FUNCTION_BLOCK FB_ReversingSequence EXTENDS FB_CyclicFB IMPLEMENTS I_MotionSequence
VAR
	_Axis		 : I_BasicAxis;
	_Position1	 : LREAL;
	_Position2	 : LREAL;
	_Velocity	 : LREAL;
	_IdleTime	 : INT;
	fbMove		 : MC_MoveAbsolute;
	fbIdle		 : TON;
	SequenceStep : E_RevSeq;
END_VAR

{warning 'add property implementation'}
PROPERTY Axis : SPT_Motion_Control.I_BasicAxis
GET
Axis := _Axis;
END_GET
SET
_Axis := Axis;
END_SET
END_PROPERTY

{warning 'add method implementation '}
METHOD CyclicLogic
CASE SequenceStep OF
	E_RevSeq.Stopped: //Idle, waiting for Execute method
	E_RevSeq.Move1:	  //Move to Position 1
		fbMove(Axis		:= _Axis.Axis,
			   Execute	:= TRUE,
			   Position := _Position1,
			   Velocity := _Velocity);

		SequenceStep := E_RevSeq.Wait1;

	E_RevSeq.Wait1:
		fbMove(Axis := _Axis.Axis, Execute := FALSE);
		IF NOT fbmove.Busy THEN
			IF NOT fbMove.Error THEN
				SequenceStep := E_RevSeq.Idle1;
			ELSE
				_ErrorID	 := 11;
				SequenceStep := E_RevSeq.Error;
			END_IF
		END_IF

	E_RevSeq.Idle1: //Wait for idle time
		fbIdle(IN := TRUE, PT := TO_TIME(_IdleTime));
		IF fbIdle.Q THEN
			fbIdle(IN := FALSE);
			SequenceStep := E_RevSeq.Move2;
		END_IF

	E_RevSeq.Move2: //Move to Posotion 2
		fbMove(Axis		:= _Axis.Axis,
			   Execute	:= TRUE,
			   Position := _Position2,
			   Velocity := _Velocity);

		SequenceStep := E_RevSeq.Wait2;

	E_RevSeq.Wait2:
		fbMove(Axis := _Axis.Axis, Execute := FALSE);
		IF NOT fbmove.Busy THEN
			IF NOT fbMove.Error THEN
				SequenceStep := E_RevSeq.Idle2;
			ELSE
				_ErrorID	 := 11;
				SequenceStep := E_RevSeq.Error;
			END_IF
		END_IF

	E_RevSeq.Idle2: //Wait for Idle time
		fbIdle(IN := TRUE, PT := TO_TIME(_IdleTime));
		IF fbIdle.Q THEN
			fbIdle(IN := FALSE);
			SequenceStep := E_RevSeq.Move1;
		END_IF

	E_RevSeq.Error: //Error Step
		_Error := TRUE;
END_CASE

_Busy := SequenceStep <> 0;
END_METHOD

{warning 'add method implementation '}
METHOD Execute : BOOL
IF (_Axis = 0) OR _Busy THEN
	RETURN;
END_IF

_Busy		 := TRUE;
_Error		 := FALSE;
_ErrorID	 := 0;
SequenceStep := E_RevSeq.Move1;
Execute		 := TRUE;
END_METHOD

PROPERTY IdleTime : INT
GET
IdleTime := _IdleTime;
END_GET
SET
_IdleTime := IdleTime;
END_SET
END_PROPERTY

PROPERTY Position1 : LREAL
GET
Position1 := _Position1;
END_GET
SET
_Position1 := Position1;
END_SET
END_PROPERTY

PROPERTY Position2 : LREAL
GET
Position2 := _Position2;
END_GET
SET
_Position2 := Position2;
END_SET
END_PROPERTY

METHOD Stop : BOOL
VAR_INPUT
END_VAR
SequenceStep := E_RevSeq.Stopped;
_Axis.Stop();
Stop := TRUE;
END_METHOD

PROPERTY Velocity : LREAL
GET
Velocity := _Velocity;
END_GET
SET
_Velocity := Velocity;
END_SET
END_PROPERTY

END_FUNCTION_BLOCK

(* stored: Version 1.1.0.1, ProductVersion 3.1.4024.12
   POU FB_ReversingSequence: Id {9caf3fe3-21c0-4675-baef-5e228678bdb8}, SpecialFunc None
   Folder I_CyclicFB: Id {971a84d7-6ea4-482b-a1d5-ed542adf21c2}
   Folder I_MotionSequence: Id {27ddc1ef-906f-4502-aa86-13076f436f95}
   Property Axis: Id {e774e632-6bed-474a-a374-325b0d5252b1}
   Get Get: Id {07e1a932-df04-4ebe-934e-45351a5b26b9}
   Set Set: Id {f3b272cc-e277-4940-8448-41fb97af6d29}
   Method CyclicLogic: Id {cc4f62f5-539c-4700-a340-a403a875c94b}
   Method Execute: Id {a8de52a2-1572-4824-be8a-a9405090d682}
   Property IdleTime: Id {200a7173-147e-429e-a882-13f8ca3643b9}
   Get Get: Id {f1c502b6-5e92-42f1-a456-68dbe9967d29}
   Set Set: Id {62cf3192-b89b-4918-93e9-710af118c190}
   Property Position1: Id {9433b65f-1b4e-4ceb-ab64-28c96f2b2fd9}
   Get Get: Id {d6713a58-aa0d-4560-87d5-6bb1ef3efc65}
   Set Set: Id {f0c49669-6992-4e27-9c4c-eda1eef605b6}
   Property Position2: Id {348dd7c4-c219-47d6-ae59-d1583256a385}
   Get Get: Id {43e72b6a-3e4d-496d-95f5-10f8c3f9e57b}
   Set Set: Id {a0bb831f-f59a-47a5-baff-143495efb4d5}
   Method Stop: Id {b61b03e4-ebb5-4472-b011-83ad31428f3d}
   Property Velocity: Id {266c92e2-1277-433c-996b-a87d45ce722c}
   Get Get: Id {09d71f05-0202-416d-93d3-84acdce3dd22}
   Set Set: Id {0eea3931-03ed-41ba-853a-869bdfc2a551} *)
